{attribute 'qualified_only'}
VAR_GLOBAL
	// Mode Selector
	bManual 			AT %I* : BOOL;
	bAuto	 			AT %I* : BOOL;
	bStartButton		AT %I* : BOOL;
	bStopButton			AT %I* : BOOL;
	
	// Raw Pressure Values
	nRawPa 				AT %I*	: INT;
	nRawPb				AT %I*	: INT;
	nRawPs				AT %I*	: INT;
	nRawPaLower			AT %I* 	: INT;
	
	// Raw Position Values
	nRawPistonPosition 	AT %I*	: INT;
	nRawJoystick		AT %I*	: INT;
	nRawFlowSensor		AT %I*	: INT;
	nRawSpoolPosition	AT %I*	: INT;
END_VAR

(* stored: Version 1.1.0.1, ProductVersion 3.1.4024.12
   GVL G_Inputs: Id {5adfdde3-399f-42d5-aa4c-f7f5d0c3a725} *)
